PROGRAM MAIN
VAR
	
END_VAR

prgLab02();
prgLab3A();
prgLab04_06();
prgLab05_07();
prgLab08();
prgLab14B();
prgLab10_11();
prgLab16();

END_PROGRAM

(* stored: Version 1.1.0.1, ProductVersion 3.1.4024.11
   POU MAIN: Id {80c62a02-491d-4597-b59c-2fe5867476c4}, SpecialFunc None *)
